FUNCTION_BLOCK F_SUB_DT_TIME (* Subtracts two number values *)
  (* Standard: 61131-3; Classification: Arithmetic; Function: SUBTRACTOR; Type: Mathematical function *)
  (* Version 1.0, 2011-09-20, 4DIAC-IDE, 4DIAC-Consortium *)
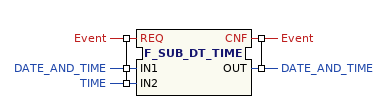
  EVENT_INPUT
    REQ WITH IN1, IN2; (* Normal Execution Request *)
  END_EVENT
  EVENT_OUTPUT
    CNF WITH OUT; (* Execution Confirmation *)
  END_EVENT
  VAR_INPUT
    IN1 : DATE_AND_TIME; (* First funtion input *)
    IN2 : TIME; (* Second function input *)
  END_VAR
  VAR_OUTPUT
    OUT : DATE_AND_TIME; (* Function output *)
  END_VAR
END_FUNCTION_BLOCK
